TYPE AdsSymbolUploadInfo2 :
STRUCT
   nSymbols : UDINT;
   nSymSize : UDINT;
   nDatatypes : UDINT;
   nDatatypeSize : UDINT;
   nMaxDynSymbols : UDINT;
   nUsedDynSymbols : UDINT;
END_STRUCT
END_TYPE

(* stored: Version 1.1.0.1, ProductVersion 3.1.4024.3
   DUT AdsSymbolUploadInfo2: Id {41b603a5-cd48-40ec-b064-b6242065875b} *)
